% RSLogix 500 project PV2.RSS, saved by version 8.30.00.16 %
PROJECT "PV2"    % processor: Bul.1763 MicroLogix 1100 Series B %

PROGRAM FILES
  LAD 2   22 rungs

DATA FILES
  O0 OUTPUT  5 elements
  I1 INPUT  7 elements
  S2 STATUS  66 elements
  B3 BINARY  3 elements
  T4 TIMER  2 elements
  C5 COUNTER  1 elements
  R6 CONTROL  1 elements
  N7 INTEGER  1 elements
  F8 FLOAT  1 elements

LADDER 2
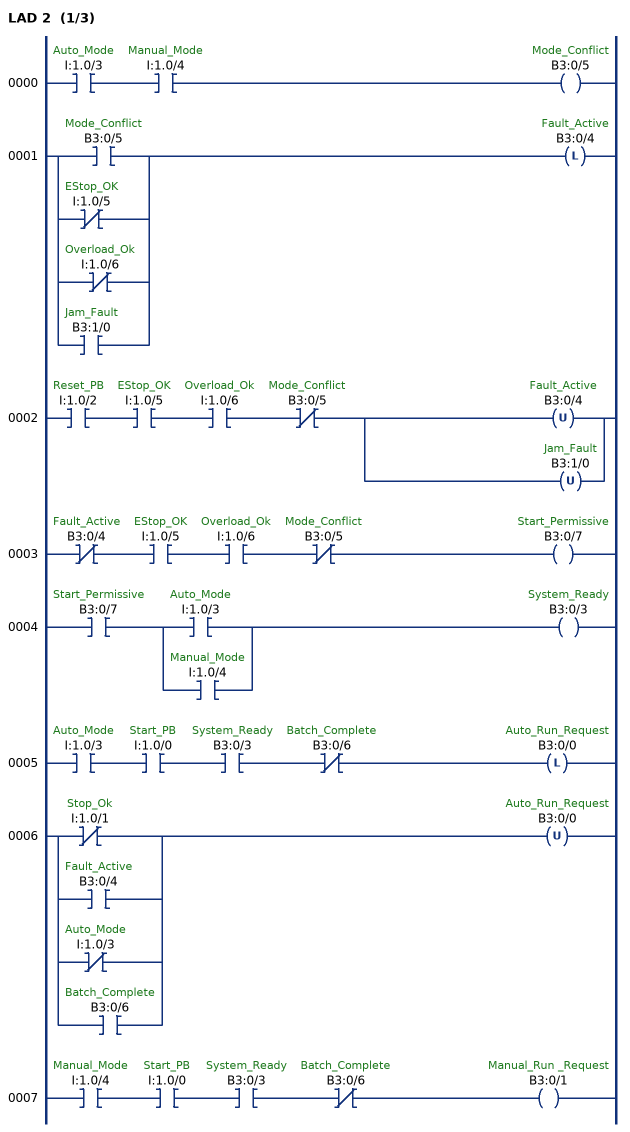
% Rung: 0 %
SOR XIC I:1.0/3 XIC I:1.0/4 OTE B3:0/5 EOR
%   I:1.0/3  "Auto_Mode" %
%   I:1.0/4  "Manual_Mode" %
%   B3:0/5  "Mode_Conflict" %
% Rung: 1 %
SOR BST XIC B3:0/5 NXB BST XIO I:1.0/5 NXB BST XIO I:1.0/6 NXB XIC B3:1/0 BND BND BND OTL B3:0/4 EOR
%   B3:0/5  "Mode_Conflict" %
%   I:1.0/5  "EStop_OK" %
%   I:1.0/6  "Overload_Ok" %
%   B3:1/0  "Jam_Fault" %
%   B3:0/4  "Fault_Active" %
% Rung: 2 %
SOR XIC I:1.0/2 XIC I:1.0/5 XIC I:1.0/6 XIO B3:0/5 BST OTU B3:0/4 NXB OTU B3:1/0 BND EOR
%   I:1.0/2  "Reset_PB" %
%   I:1.0/5  "EStop_OK" %
%   I:1.0/6  "Overload_Ok" %
%   B3:0/5  "Mode_Conflict" %
%   B3:0/4  "Fault_Active" %
%   B3:1/0  "Jam_Fault" %
% Rung: 3 %
SOR XIO B3:0/4 XIC I:1.0/5 XIC I:1.0/6 XIO B3:0/5 OTE B3:0/7 EOR
%   B3:0/4  "Fault_Active" %
%   I:1.0/5  "EStop_OK" %
%   I:1.0/6  "Overload_Ok" %
%   B3:0/5  "Mode_Conflict" %
%   B3:0/7  "Start_Permissive" %
% Rung: 4 %
SOR XIC B3:0/7 BST XIC I:1.0/3 NXB XIC I:1.0/4 BND OTE B3:0/3 EOR
%   B3:0/7  "Start_Permissive" %
%   I:1.0/3  "Auto_Mode" %
%   I:1.0/4  "Manual_Mode" %
%   B3:0/3  "System_Ready" %
% Rung: 5 %
SOR XIC I:1.0/3 XIC I:1.0/0 XIC B3:0/3 XIO B3:0/6 OTL B3:0/0 EOR
%   I:1.0/3  "Auto_Mode" %
%   I:1.0/0  "Start_PB" %
%   B3:0/3  "System_Ready" %
%   B3:0/6  "Batch_Complete" %
%   B3:0/0  "Auto_Run_Request" %
% Rung: 6 %
SOR BST XIO I:1.0/1 NXB BST XIC B3:0/4 NXB BST XIO I:1.0/3 NXB XIC B3:0/6 BND BND BND OTU B3:0/0 EOR
%   I:1.0/1  "Stop_Ok" %
%   B3:0/4  "Fault_Active" %
%   I:1.0/3  "Auto_Mode" %
%   B3:0/6  "Batch_Complete" %
%   B3:0/0  "Auto_Run_Request" %
% Rung: 7 %
SOR XIC I:1.0/4 XIC I:1.0/0 XIC B3:0/3 XIO B3:0/6 OTE B3:0/1 EOR
%   I:1.0/4  "Manual_Mode" %
%   I:1.0/0  "Start_PB" %
%   B3:0/3  "System_Ready" %
%   B3:0/6  "Batch_Complete" %
%   B3:0/1  "Manual_Run _Request" %

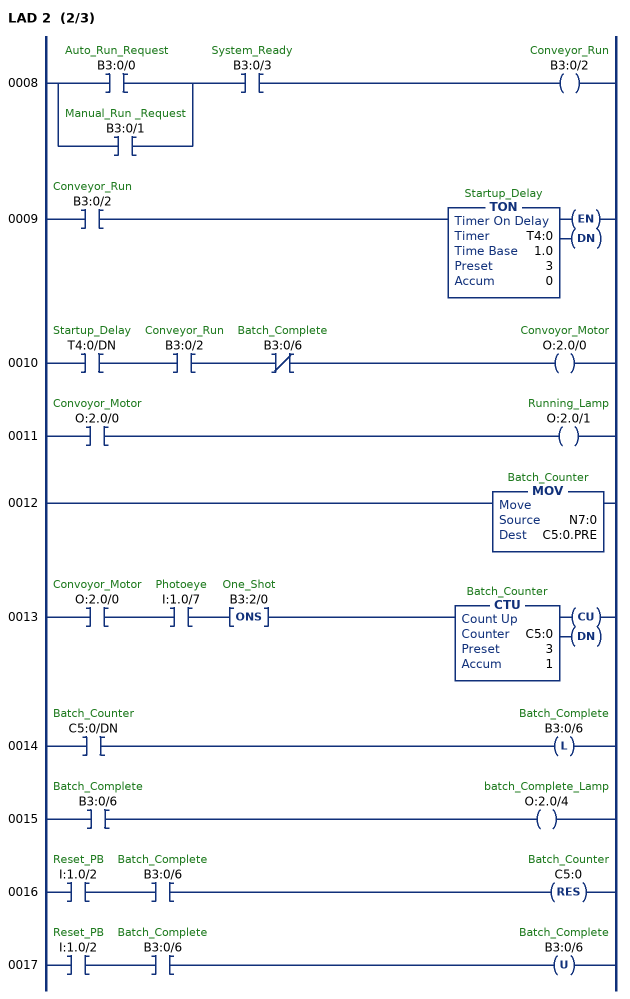
% Rung: 8 %
SOR BST XIC B3:0/0 NXB XIC B3:0/1 BND XIC B3:0/3 OTE B3:0/2 EOR
%   B3:0/0  "Auto_Run_Request" %
%   B3:0/1  "Manual_Run _Request" %
%   B3:0/3  "System_Ready" %
%   B3:0/2  "Conveyor_Run" %
% Rung: 9 %
SOR XIC B3:0/2 TON T4:0 1.0 3 0 EOR
%   B3:0/2  "Conveyor_Run" %
%   T4:0  "Startup_Delay" %
% Rung: 10 %
SOR XIC T4:0/DN XIC B3:0/2 XIO B3:0/6 OTE O:2.0/0 EOR
%   T4:0  "Startup_Delay" %
%   B3:0/2  "Conveyor_Run" %
%   B3:0/6  "Batch_Complete" %
%   O:2.0/0  "Convoyor_Motor" %
% Rung: 11 %
SOR XIC O:2.0/0 OTE O:2.0/1 EOR
%   O:2.0/0  "Convoyor_Motor" %
%   O:2.0/1  "Running_Lamp" %
% Rung: 12 %
SOR MOV N7:0 C5:0.PRE EOR
%   C5:0  "Batch_Counter" %
% Rung: 13 %
SOR XIC O:2.0/0 XIC I:1.0/7 ONS B3:2/0 CTU C5:0 3 1 EOR
%   O:2.0/0  "Convoyor_Motor" %
%   I:1.0/7  "Photoeye" %
%   B3:2/0  "One_Shot" %
%   C5:0  "Batch_Counter" %
% Rung: 14 %
SOR XIC C5:0/DN OTL B3:0/6 EOR
%   C5:0  "Batch_Counter" %
%   B3:0/6  "Batch_Complete" %
% Rung: 15 %
SOR XIC B3:0/6 OTE O:2.0/4 EOR
%   B3:0/6  "Batch_Complete" %
%   O:2.0/4  "batch_Complete_Lamp" %
% Rung: 16 %
SOR XIC I:1.0/2 XIC B3:0/6 RES C5:0 EOR
%   I:1.0/2  "Reset_PB" %
%   B3:0/6  "Batch_Complete" %
%   C5:0  "Batch_Counter" %
% Rung: 17 %
SOR XIC I:1.0/2 XIC B3:0/6 OTU B3:0/6 EOR
%   I:1.0/2  "Reset_PB" %
%   B3:0/6  "Batch_Complete" %

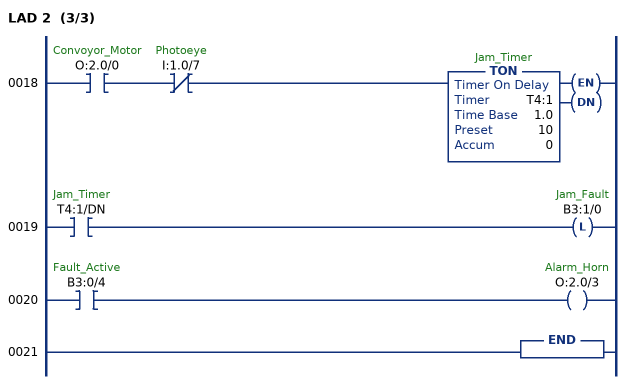
% Rung: 18 %
SOR XIC O:2.0/0 XIO I:1.0/7 TON T4:1 1.0 10 0 EOR
%   O:2.0/0  "Convoyor_Motor" %
%   I:1.0/7  "Photoeye" %
%   T4:1  "Jam_Timer" %
% Rung: 19 %
SOR XIC T4:1/DN OTL B3:1/0 EOR
%   T4:1  "Jam_Timer" %
%   B3:1/0  "Jam_Fault" %
% Rung: 20 %
SOR XIC B3:0/4 OTE O:2.0/3 EOR
%   B3:0/4  "Fault_Active" %
%   O:2.0/3  "Alarm_Horn" %
% Rung: 21 %
SOR END EOR

OTHER DOCUMENTED ADDRESSES
  B3:1/1  "Mode_Fault"
  B3:1/2  "EStop_Fault"
  B3:1/3  "Overload_Fault"
  I:0.0/2  "Reset_PB"
  I:0.0/3  "Auto_Mode"
  I:0.0/4  "Manual_Mode"
  I:0.0/5  "EStop_OK"
  I:0.0/6  "Overload_OK"
  I:5  "EStop_Ok"

DATA TABLE (non-zero values as saved)
DATA B3
% B3:0 % 0X0010 0X0001 0X0000
DATA T4
% .PRE .ACC %
% T4:0 % 3 0
% T4:1 % 10 0
DATA C5
% .PRE .ACC %
% C5:0 % 3 1
DATA N7
% N7:0 % 3
